(* CoDeSys 2.3.9.42 project: A100-60_CR0020_V050003.pro *)
(* Libraries: ifm_CR0020\ifm_CR0020_V050003.lib 15.12.08 18:14:24, Util.lib 6.11.07 15:39:24, standard.lib 4.10.05 11:14:46, ifm_J1939\ifm_CAN1_EXT_V050008.lib 12.9.08 16:16:28, ifm_J1939\ifm_J1939_1_V050008.lib 5.2.08 18:55:26, ifm_J1939\ifm_J1939_2_V050008.lib 5.2.08 18:56:24 *)

(* PLC configuration (modules and I/O channels)
Inputs Port0 [Eingangsport0] node 0, in %IB0 out %QB0
  I00 AT %IX0.0 [BoolChannelIn] Connector 1, Pin 08, (see Configuration Byte I00_MODE)
  I01 AT %IX0.1 [BoolChannelIn] Connector 1, Pin 27, (see Configuration Byte I01_MODE)
  I02 AT %IX0.2 [BoolChannelIn] Connector 1, Pin 09, (see Configuration Byte I02_MODE)
  I03 AT %IX0.3 [BoolChannelIn] Connector 1, Pin 28, (see Configuration Byte I03_MODE)
  I04 AT %IX0.4 [BoolChannelIn] Connector 1, Pin 10, (see Configuration Byte I04_MODE)
  I05 AT %IX0.5 [BoolChannelIn] Connector 1, Pin 29, (see Configuration Byte I05_MODE)
  I06 AT %IX0.6 [BoolChannelIn] Connector 1, Pin 11, (see Configuration Byte I06_MODE)
  I07 AT %IX0.7 [BoolChannelIn] Connector 1, Pin 30, (see Configuration Byte I07_MODE)
Inputs Port1 [Eingangsport1] node 0, in %IB1 out %QB0
  I10 AT %IX0.8 [BoolChannelIn] Connector 1, Pin 44, (see Configuration Byte I10_MODE)
  I11 AT %IX0.9 [BoolChannelIn] Connector 1, Pin 45, (see Configuration Byte I11_MODE)
  I12 AT %IX0.10 [BoolChannelIn] Connector 1, Pin 46, (see Configuration Byte I12_MODE)
  I13 AT %IX0.11 [BoolChannelIn] Connector 1, Pin 47, (see Configuration Byte I13_MODE)
  I14 AT %IX0.12 [BoolChannelIn] Connector 1, Pin 20, (see Configuration Byte I14_MODE)
  I15 AT %IX0.13 [BoolChannelIn] Connector 1, Pin 02, (see Configuration Byte I15_MODE)
  I16 AT %IX0.14 [BoolChannelIn] Connector 1, Pin 21, (see Configuration Byte I16_MODE)
  I17 AT %IX0.15 [BoolChannelIn] Connector 1, Pin 38, (see Configuration Byte I17_MODE)
Inputs Port2 [Eingangsport2] node 0, in %IB2 out %QB0
  I20 AT %IX1.0 [BoolChannelIn] Connector 1, Pin 36, (see Configuration Byte I20_MODE)
  I21 AT %IX1.1 [BoolChannelIn] Connector 1, Pin 54, (see Configuration Byte I21_MODE)
  I22 AT %IX1.2 [BoolChannelIn] Connector 1, Pin 17, (see Configuration Byte I22_MODE)
  I23 AT %IX1.3 [BoolChannelIn] Connector 1, Pin 53, (see Configuration Byte I23_MODE)
  I24 AT %IX1.4 [BoolChannelIn] Connector 1, Pin 19, (see Configuration Byte I24_MODE)
  I25 AT %IX1.5 [BoolChannelIn] Connector 1, Pin 55, (see Configuration Byte I25_MODE)
  I26 AT %IX1.6 [BoolChannelIn] Connector 1, Pin 18, (see Configuration Byte I26_MODE)
  I27 AT %IX1.7 [BoolChannelIn] Connector 1, Pin 37, (see Configuration Byte I27_MODE)
Inputs Port3 [Eingangsport3] node 0, in %IB3 out %QB0
  I30 AT %IX1.8 [BoolChannelIn] Connector 1, Pin 39, (see Configuration Byte I30_MODE)
  I31 AT %IX1.9 [BoolChannelIn] Connector 1, Pin 03, (see Configuration Byte I31_MODE)
  I32 AT %IX1.10 [BoolChannelIn] Connector 1, Pin 40, (see Configuration Byte I32_MODE)
  I33 AT %IX1.11 [BoolChannelIn] Connector 1, Pin 22, (see Configuration Byte I33_MODE)
  I34 AT %IX1.12 [BoolChannelIn] Connector 1, Pin 41, (see Configuration Byte I34_MODE)
  I35 AT %IX1.13 [BoolChannelIn] Connector 1, Pin 42, (see Configuration Byte I35_MODE)
  I36 AT %IX1.14 [BoolChannelIn] Connector 1, Pin 43, (see Configuration Byte I36_MODE)
  I37 AT %IX1.15 [BoolChannelIn] Connector 1, Pin 04, (see Configuration Byte I37_MODE)
Inputs Port4 [Eingangsport4] node 0, in %IB4 out %QB0
  I40 AT %IX2.0 [BoolChannelIn] Connector 1, Pin 48, (see Configuration Byte I40_MODE)
  I41 AT %IX2.1 [BoolChannelIn] Connector 1, Pin 49, (see Configuration Byte I41_MODE)
  I42 AT %IX2.2 [BoolChannelIn] Connector 1, Pin 31, (see Configuration Byte I42_MODE)
  I43 AT %IX2.3 [BoolChannelIn] Connector 1, Pin 50, (see Configuration Byte I43_MODE)
  I44 AT %IX2.4 [BoolChannelIn] Connector 1, Pin 51, (see Configuration Byte I44_MODE)
  I45 AT %IX2.5 [BoolChannelIn] Connector 1, Pin 52, (see Configuration Byte I45_MODE)
  I46 AT %IX2.6 [BoolChannelIn] Connector 1, Pin 16, (see Configuration Byte I46_MODE)
  I47 AT %IX2.7 [BoolChannelIn] Connector 1, Pin 35, (see Configuration Byte I47_MODE)
ANALOG0 AT %IW3 [WordChannelIn] Connector 1, Pin 08, ANALOG CHANNEL 0
ANALOG1 AT %IW4 [WordChannelIn] Connector 1, Pin 27, ANALOG CHANNEL 1
ANALOG2 AT %IW5 [WordChannelIn] Connector 1, Pin 09, ANALOG CHANNEL 2
ANALOG3 AT %IW6 [WordChannelIn] Connector 1, Pin 28, ANALOG CHANNEL 3
ANALOG4 AT %IW7 [WordChannelIn] Connector 1, Pin 10, ANALOG CHANNEL 4
ANALOG5 AT %IW8 [WordChannelIn] Connector 1, Pin 29, ANALOG CHANNEL 5
ANALOG6 AT %IW9 [WordChannelIn] Connector 1, Pin 11, ANALOG CHANNEL 6
ANALOG7 AT %IW10 [WordChannelIn] Connector 1, Pin 30, ANALOG CHANNEL 7
Inputs Miscellaneous [Eingaenge] node 0, in %IB22 out %QB0
  SUPPLY_VOLTAGE AT %IW11 [WordChannelIn] SUPPLY VOLTAGE
  CLAMP_15 AT %IX12.0 [WordChannelIn] CLAMP 15
Outputs Port1 [Ausgangsport1] node 0, in %IB64 out %QB0
  Q10 AT %QX0.0 [BoolChannelOut] Connector 1, Pin 44, (see Configuration Byte Q10_MODE)
  Q11 AT %QX0.1 [BoolChannelOut] Connector 1, Pin 45, (see Configuration Byte Q11_MODE)
  Q12 AT %QX0.2 [BoolChannelOut] Connector 1, Pin 46, (see Configuration Byte Q12_MODE)
  Q13 AT %QX0.3 [BoolChannelOut] Connector 1, Pin 47, (see Configuration Byte Q13_MODE)
Outputs Port2 [Ausgangsport2] node 0, in %IB64 out %QB0
  Q20 AT %QX0.4 [BoolChannelOut] Connector 1, Pin 36, (see Configuration Byte Q20_MODE)
  Q21 AT %QX0.5 [BoolChannelOut] Connector 1, Pin 54, (see Configuration Byte Q21_MODE)
  Q22 AT %QX0.6 [BoolChannelOut] Connector 1, Pin 17, (see Configuration Byte Q22_MODE)
  Q23 AT %QX0.7 [BoolChannelOut] Connector 1, Pin 53, (see Configuration Byte Q23_MODE)
Outputs Port3 [Ausgangsport3] node 0, in %IB64 out %QB1
  Q30 AT %QX0.8 [BoolChannelOut] Connector 1, Pin 39, (see Configuration Byte Q30_MODE)
  Q31 AT %QX0.9 [BoolChannelOut] Connector 1, Pin 03, (see Configuration Byte Q31_MODE)
  Q32 AT %QX0.10 [BoolChannelOut] Connector 1, Pin 40, (see Configuration Byte Q32_MODE)
  Q33 AT %QX0.11 [BoolChannelOut] Connector 1, Pin 22, (see Configuration Byte Q33_MODE)
  Q34 AT %QX0.12 [BoolChannelOut] Connector 1, Pin 41, (see Configuration Byte Q34_MODE)
  Q35 AT %QX0.13 [BoolChannelOut] Connector 1, Pin 42, (see Configuration Byte Q35_MODE)
  Q36 AT %QX0.14 [BoolChannelOut] Connector 1, Pin 43, (see Configuration Byte Q36_MODE)
  Q37 AT %QX0.15 [BoolChannelOut] Connector 1, Pin 04, (see Configuration Byte Q37_MODE)
Outputs Port4 [Ausgangsport4] node 0, in %IB64 out %QB2
  Q40 AT %QX1.0 [BoolChannelOut] Connector 1, Pin 48, (see Configuration Byte Q40_MODE)
  Q41 AT %QX1.1 [BoolChannelOut] Connector 1, Pin 49, (see Configuration Byte Q41_MODE)
  Q42 AT %QX1.2 [BoolChannelOut] Connector 1, Pin 31, (see Configuration Byte Q42_MODE)
  Q43 AT %QX1.3 [BoolChannelOut] Connector 1, Pin 50, (see Configuration Byte Q43_MODE)
  Q44 AT %QX1.4 [BoolChannelOut] Connector 1, Pin 51, (see Configuration Byte Q44_MODE)
  Q45 AT %QX1.5 [BoolChannelOut] Connector 1, Pin 52, (see Configuration Byte Q45_MODE)
  Q46 AT %QX1.6 [BoolChannelOut] Connector 1, Pin 16, (see Configuration Byte Q46_MODE)
  Q47 AT %QX1.7 [BoolChannelOut] Connector 1, Pin 35, (see Configuration Byte Q47_MODE)
Input Modes Port0 [EingangsModi0] node 0, in %IB64 out %QB8
  I00_MODE AT %QB8 [ByteChannelOut] Configuration Byte for Input Pin 08, Connector 1
  I01_MODE AT %QB9 [ByteChannelOut] Configuration Byte for Input Pin 27, Connector 1
  I02_MODE AT %QB10 [ByteChannelOut] Configuration Byte for Input Pin 09, Connector 1
  I03_MODE AT %QB11 [ByteChannelOut] Configuration Byte for Input Pin 28, Connector 1
  I04_MODE AT %QB12 [ByteChannelOut] Configuration Byte for Input Pin 10, Connector 1
  I05_MODE AT %QB13 [ByteChannelOut] Configuration Byte for Input Pin 29, Connector 1
  I06_MODE AT %QB14 [ByteChannelOut] Configuration Byte for Input Pin 11, Connector 1
  I07_MODE AT %QB15 [ByteChannelOut] Configuration Byte for Input Pin 30, Connector 1
Input Modes Port1 [EingangsModi1] node 0, in %IB64 out %QB16
  I14_MODE AT %QB16 [ByteChannelOut] Configuration Byte for Input Pin 20, Connector 1
  I15_MODE AT %QB17 [ByteChannelOut] Configuration Byte for Input Pin 02, Connector 1
  I16_MODE AT %QB18 [ByteChannelOut] Configuration Byte for Input Pin 21, Connector 1
  I17_MODE AT %QB19 [ByteChannelOut] Configuration Byte for Input Pin 38, Connector 1
Input Modes Port2 [EingangsModi2] node 0, in %IB64 out %QB20
  I24_MODE AT %QB20 [ByteChannelOut] Configuration Byte for Input Pin 19, Connector 1
  I25_MODE AT %QB21 [ByteChannelOut] Configuration Byte for Input Pin 55, Connector 1
  I26_MODE AT %QB22 [ByteChannelOut] Configuration Byte for Input Pin 18, Connector 1
  I27_MODE AT %QB23 [ByteChannelOut] Configuration Byte for Input Pin 37, Connector 1
Input Modes Port3 [EingangsModi3] node 0, in %IB64 out %QB24
  I30_MODE AT %QB24 [ByteChannelOut] Configuration Byte for Input Pin 39, Connector 1
  I31_MODE AT %QB25 [ByteChannelOut] Configuration Byte for Input Pin 03, Connector 1
  I32_MODE AT %QB26 [ByteChannelOut] Configuration Byte for Input Pin 40, Connector 1
  I33_MODE AT %QB27 [ByteChannelOut] Configuration Byte for Input Pin 22, Connector 1
  I34_MODE AT %QB28 [ByteChannelOut] Configuration Byte for Input Pin 41, Connector 1
  I35_MODE AT %QB29 [ByteChannelOut] Configuration Byte for Input Pin 42, Connector 1
  I36_MODE AT %QB30 [ByteChannelOut] Configuration Byte for Input Pin 43, Connector 1
  I37_MODE AT %QB31 [ByteChannelOut] Configuration Byte for Input Pin 04, Connector 1
Input Modes Port4 [EingangsModi4] node 0, in %IB64 out %QB32
  I40_MODE AT %QB32 [ByteChannelOut] Configuration Byte for Input Pin 48, Connector 1
  I41_MODE AT %QB33 [ByteChannelOut] Configuration Byte for Input Pin 49, Connector 1
  I42_MODE AT %QB34 [ByteChannelOut] Configuration Byte for Input Pin 31, Connector 1
  I43_MODE AT %QB35 [ByteChannelOut] Configuration Byte for Input Pin 50, Connector 1
  I44_MODE AT %QB36 [ByteChannelOut] Configuration Byte for Input Pin 51, Connector 1
  I45_MODE AT %QB37 [ByteChannelOut] Configuration Byte for Input Pin 52, Connector 1
  I46_MODE AT %QB38 [ByteChannelOut] Configuration Byte for Input Pin 16, Connector 1
  I47_MODE AT %QB39 [ByteChannelOut] Configuration Byte for Input Pin 35, Connector 1
Output Modes Port1 [AusgangsModi1] node 0, in %IB64 out %QB40
  Q10_MODE AT %QB40 [ByteChannelOut] Configuration Byte for Output Pin 44, Connector 1
  Q11_MODE AT %QB41 [ByteChannelOut] Configuration Byte for Output Pin 45, Connector 1
  Q12_MODE AT %QB42 [ByteChannelOut] Configuration Byte for Output Pin 46, Connector 1
  Q13_MODE AT %QB43 [ByteChannelOut] Configuration Byte for Output Pin 47, Connector 1
Output Modes Port2 [AusgangsModi2] node 0, in %IB64 out %QB44
  Q20_MODE AT %QB44 [ByteChannelOut] Configuration Byte for Output Pin 36, Connector 1
  Q21_MODE AT %QB45 [ByteChannelOut] Configuration Byte for Output Pin 54, Connector 1
  Q22_MODE AT %QB46 [ByteChannelOut] Configuration Byte for Output Pin 17, Connector 1
  Q23_MODE AT %QB47 [ByteChannelOut] Configuration Byte for Output Pin 53, Connector 1
Output Modes Port3 [AusgangsModi3] node 0, in %IB64 out %QB48
  Q30_MODE AT %QB48 [ByteChannelOut] Configuration Byte for Output Pin 39, Connector 1
  Q31_MODE AT %QB49 [ByteChannelOut] Configuration Byte for Output Pin 03, Connector 1
  Q32_MODE AT %QB50 [ByteChannelOut] Configuration Byte for Output Pin 40, Connector 1
  Q33_MODE AT %QB51 [ByteChannelOut] Configuration Byte for Output Pin 22, Connector 1
  Q34_MODE AT %QB52 [ByteChannelOut] Configuration Byte for Output Pin 41, Connector 1
  Q35_MODE AT %QB53 [ByteChannelOut] Configuration Byte for Output Pin 42, Connector 1
  Q36_MODE AT %QB54 [ByteChannelOut] Configuration Byte for Output Pin 43, Connector 1
  Q37_MODE AT %QB55 [ByteChannelOut] Configuration Byte for Output Pin 04, Connector 1
Output Modes Port4 [AusgangsModi4] node 0, in %IB64 out %QB56
  Q40_MODE AT %QB56 [ByteChannelOut] Configuration Byte for Output Pin 48, Connector 1
  Q41_MODE AT %QB57 [ByteChannelOut] Configuration Byte for Output Pin 49, Connector 1
  Q42_MODE AT %QB58 [ByteChannelOut] Configuration Byte for Output Pin 31, Connector 1
  Q43_MODE AT %QB59 [ByteChannelOut] Configuration Byte for Output Pin 50, Connector 1
  Q44_MODE AT %QB60 [ByteChannelOut] Configuration Byte for Output Pin 51, Connector 1
  Q45_MODE AT %QB61 [ByteChannelOut] Configuration Byte for Output Pin 52, Connector 1
  Q46_MODE AT %QB62 [ByteChannelOut] Configuration Byte for Output Pin 16, Connector 1
  Q47_MODE AT %QB63 [ByteChannelOut] Configuration Byte for Output Pin 35, Connector 1
*)

(* Global variable list: GV_CAL *)
VAR_GLOBAL
(*
	Аналоговый - aChannel_ADC - adc := 0 - 16
	Частотный  - aChannel_PIN - pin := 1 - 8
	ШИМ        - aChannel_PWM - pwm := 2 - 8
	ПИД        - aChannel_PID - pid := 3 - 8
	Энкодер    - aChannel_ENC - enc := 4 - 8
	Расчет     - aChannel_FRM - frm := 5 - 8
	Расход                          := 6 - 8
*)

(*Максимальный размер массива параметров каналов*)
	iSizeArrayParamMax : INT := 64;

(**)
	aPage_Channel      : ARRAY [0..63] OF Page_Channel;(**)

(*Переменные выбора текущего режима работы*)
	dwCurrMode         : DWORD := 1;(*Текущий режим работы установки*)
	bCurrModeChange    : BOOL  := 0;(*Флаг смены текущего режима работы установки*)

(*Переменные каналов ШИМ*)
	rArrayDataPWM_XH      : ARRAY [1..8] OF REAL;(**)
	rArrayDataPWM_XL      : ARRAY [1..8] OF REAL;(**)
	rArrayDataPWM_YH      : ARRAY [1..8] OF REAL;(**)
	rArrayDataPWM_YL      : ARRAY [1..8] OF REAL;(**)
	dwArrayAverTimePWM    : ARRAY [1..8] OF DWORD;(*Времена усреднения каналов*)
	rArrayDataPWM_DZ_MAX  : ARRAY [1..8] OF REAL;(*Коэффициенты, учитывающие особенности механики*)
	dwArrayDataPWM_DZ_MIN : ARRAY [1..8] OF DWORD;(**)

	dwArrayNumberPWM      : ARRAY [1..8] OF DWORD;(**)
	rArrayParam10PWM      : ARRAY [1..8] OF REAL;(**)

(*Переменные каналов ПИД*)
	rArrayDataPID_P_Coef  : ARRAY [1..8] OF REAL;(**)
	rArrayDataPID_I_Coef  : ARRAY [1..8] OF REAL;(**)
	rArrayDataPID_D_Coef  : ARRAY [1..8] OF REAL;(**)
	rArrayDataPID_Shift   : ARRAY [1..8] OF REAL;(**)
	dwArrayAverTimePID    : ARRAY [1..8] OF DWORD;(*Времена усреднения каналов*)
	rArrayCoeffPID        : ARRAY [1..8] OF REAL;(*Коэффициенты, учитывающие особенности механики*)
	dwArrayDescriptPID    : ARRAY [1..8] OF DWORD;(**)

	dwArrayNumberPID      : ARRAY [1..8] OF DWORD;(**)
	rArrayParam10PID      : ARRAY [1..8] OF REAL;(**)
END_VAR

(* Global variable list: GV_CAN1_J1939 *)
VAR_GLOBAL
(*Переменные параметров CAN шины*)
	byCAN1_PCUnitID            : BYTE := 16#01;(*ID компьютерной панели, подключенной на CAN1*)

	byCAN1_DownloadID          : BYTE := 127;(*ID контроллера CAN1 (Download)*)
	byCAN1_PreferAddr          : BYTE := 16#40;(**)             byCurrCAN1Addr   : BYTE;(*Текущий адрес на шине CAN PC*)
	byCAN1_Channel             : BYTE := 1;
	byCAN1_DataLength          : BYTE := 8;(*Количество байт в пакете CAN1*)
	wCAN1_BaudRate             : WORD := 250;(*Скорость передачи данных 250 кбит/сек*)
	bCAN1_TransmitEnable       : BOOL := 1;(*Разрешение работы CAN1 на передачу*)

	bCAN1_J1939NotActive       : BOOL := 0;(*CAN J1939 Not active*)
	bCAN1_J1939Errors          : BOOL := 0;(*CAN J1939 Signalling of errors*)

(*Переменные приема в CAN J1939*)
	CAN1RX_UNIT_ADDR           : J1939_1_RECEIVE;  abyCAN1RX_UNIT_ADDR           : ARRAY [0..7] OF BYTE;

	CAN1RX_CHANNEL_INDEX       : J1939_1_RECEIVE;  abyCAN1RX_CHANNEL_INDEX       : ARRAY [0..7] OF BYTE;
	CAN1RX_PARAM00             : J1939_1_RECEIVE;  abyCAN1RX_PARAM00             : ARRAY [0..7] OF BYTE;
	CAN1RX_PARAM01             : J1939_1_RECEIVE;  abyCAN1RX_PARAM01             : ARRAY [0..7] OF BYTE;
	CAN1RX_PARAM02             : J1939_1_RECEIVE;  abyCAN1RX_PARAM02             : ARRAY [0..7] OF BYTE;
	CAN1RX_PARAM03             : J1939_1_RECEIVE;  abyCAN1RX_PARAM03             : ARRAY [0..7] OF BYTE;
	CAN1RX_PARAM04             : J1939_1_RECEIVE;  abyCAN1RX_PARAM04             : ARRAY [0..7] OF BYTE;
	CAN1RX_PARAM05             : J1939_1_RECEIVE;  abyCAN1RX_PARAM05             : ARRAY [0..7] OF BYTE;
	CAN1RX_PARAM06             : J1939_1_RECEIVE;  abyCAN1RX_PARAM06             : ARRAY [0..7] OF BYTE;
	CAN1RX_PARAM07             : J1939_1_RECEIVE;  abyCAN1RX_PARAM07             : ARRAY [0..7] OF BYTE;
	CAN1RX_PARAM08             : J1939_1_RECEIVE;  abyCAN1RX_PARAM08             : ARRAY [0..7] OF BYTE;
	CAN1RX_PARAM09             : J1939_1_RECEIVE;  abyCAN1RX_PARAM09             : ARRAY [0..7] OF BYTE;
	CAN1RX_PARAM10             : J1939_1_RECEIVE;  abyCAN1RX_PARAM10             : ARRAY [0..7] OF BYTE;

	CAN1RX_CURR_MODE           : J1939_1_RECEIVE;  abyCAN1RX_CURR_MODE           : ARRAY [0..7] OF BYTE;
	CAN1RX_COMMAND             : J1939_1_RECEIVE;  abyCAN1RX_COMMAND             : ARRAY [0..7] OF BYTE;

	CAN1RX_Set_GN2TempManual   : J1939_1_RECEIVE;  abyCAN1RX_Set_GN2TempManual   : ARRAY [0..7] OF BYTE;
	CAN1RX_Set_GN2OverPres     : J1939_1_RECEIVE;  abyCAN1RX_Set_GN2OverPres     : ARRAY [0..7] OF BYTE;
	CAN1RX_Set_BoostPresManual : J1939_1_RECEIVE;  abyCAN1RX_Set_BoostPresManual : ARRAY [0..7] OF BYTE;
	CAN1RX_Set_GN2Rate         : J1939_1_RECEIVE;  abyCAN1RX_Set_GN2Rate         : ARRAY [0..7] OF BYTE;
	CAN1RX_Set_LN2SaturTemp    : J1939_1_RECEIVE;  abyCAN1RX_Set_LN2SaturTemp    : ARRAY [0..7] OF BYTE;

(*Переменные отправки в CAN J1939. Используемые PGN*)
	CAN1TX_UNIT_ADDR           : J1939_1_TRANSMIT; abyCAN1TX_UNIT_ADDR           : ARRAY [0..7] OF BYTE; dwPGN1_UNIT_ADDR           : DWORD := 16#F000;

	CAN1TX_CHANNEL_INDEX       : J1939_1_TRANSMIT; abyCAN1TX_CHANNEL_INDEX       : ARRAY [0..7] OF BYTE; dwPGN1_CHANNEL_INDEX       : DWORD := 16#F001;
	CAN1TX_PARAM00             : J1939_1_TRANSMIT; abyCAN1TX_PARAM00             : ARRAY [0..7] OF BYTE; dwPGN1_PARAM00             : DWORD := 16#F002;
	CAN1TX_PARAM01             : J1939_1_TRANSMIT; abyCAN1TX_PARAM01             : ARRAY [0..7] OF BYTE; dwPGN1_PARAM01             : DWORD := 16#F003;
	CAN1TX_PARAM02             : J1939_1_TRANSMIT; abyCAN1TX_PARAM02             : ARRAY [0..7] OF BYTE; dwPGN1_PARAM02             : DWORD := 16#F004;
	CAN1TX_PARAM03             : J1939_1_TRANSMIT; abyCAN1TX_PARAM03             : ARRAY [0..7] OF BYTE; dwPGN1_PARAM03             : DWORD := 16#F005;
	CAN1TX_PARAM04             : J1939_1_TRANSMIT; abyCAN1TX_PARAM04             : ARRAY [0..7] OF BYTE; dwPGN1_PARAM04             : DWORD := 16#F006;
	CAN1TX_PARAM05             : J1939_1_TRANSMIT; abyCAN1TX_PARAM05             : ARRAY [0..7] OF BYTE; dwPGN1_PARAM05             : DWORD := 16#F007;
	CAN1TX_PARAM06             : J1939_1_TRANSMIT; abyCAN1TX_PARAM06             : ARRAY [0..7] OF BYTE; dwPGN1_PARAM06             : DWORD := 16#F008;
	CAN1TX_PARAM07             : J1939_1_TRANSMIT; abyCAN1TX_PARAM07             : ARRAY [0..7] OF BYTE; dwPGN1_PARAM07             : DWORD := 16#F009;
	CAN1TX_PARAM08             : J1939_1_TRANSMIT; abyCAN1TX_PARAM08             : ARRAY [0..7] OF BYTE; dwPGN1_PARAM08             : DWORD := 16#F00A;
	CAN1TX_PARAM09             : J1939_1_TRANSMIT; abyCAN1TX_PARAM09             : ARRAY [0..7] OF BYTE; dwPGN1_PARAM09             : DWORD := 16#F00B;
	CAN1TX_PARAM10             : J1939_1_TRANSMIT; abyCAN1TX_PARAM10             : ARRAY [0..7] OF BYTE; dwPGN1_PARAM10             : DWORD := 16#F00C;

	CAN1TX_CURR_MODE           : J1939_1_TRANSMIT; abyCAN1TX_CURR_MODE           : ARRAY [0..7] OF BYTE; dwPGN1_CURR_MODE           : DWORD := 16#F00D;

	CAN1TX_TOTAL_TIME          : J1939_1_TRANSMIT; abyCAN1TX_TOTAL_TIME          : ARRAY [0..7] OF BYTE; dwPGN1_TOTAL_TIME          : DWORD := 16#F00E;
	CAN1TX_LAST_TIME           : J1939_1_TRANSMIT; abyCAN1TX_LAST_TIME           : ARRAY [0..7] OF BYTE; dwPGN1_LAST_TIME           : DWORD := 16#F00F;

	CAN1TX_COMMAND             : J1939_1_TRANSMIT; abyCAN1TX_COMMAND             : ARRAY [0..7] OF BYTE; dwPGN1_COMMAND             : DWORD := 16#F010;

	CAN1TX_STATE_ADC_MS        : J1939_1_TRANSMIT; abyCAN1TX_STATE_ADC_MS        : ARRAY [0..7] OF BYTE; dwPGN1_STATE_ADC_MS        : DWORD := 16#F011;
	CAN1TX_STATE_ADC_SL1       : J1939_1_TRANSMIT; abyCAN1TX_STATE_ADC_SL1       : ARRAY [0..7] OF BYTE; dwPGN1_STATE_ADC_SL1       : DWORD := 16#F012;
	CAN1TX_STATE_ADC_SL2       : J1939_1_TRANSMIT; abyCAN1TX_STATE_ADC_SL2       : ARRAY [0..7] OF BYTE; dwPGN1_STATE_ADC_SL2       : DWORD := 16#F013;
	CAN1TX_STATE_ADC_SL3       : J1939_1_TRANSMIT; abyCAN1TX_STATE_ADC_SL3       : ARRAY [0..7] OF BYTE; dwPGN1_STATE_ADC_SL3       : DWORD := 16#F014;

	CAN1TX_MS_SV               : J1939_1_TRANSMIT; abyCAN1TX_MS_SV               : ARRAY [0..7] OF BYTE; dwPGN1_MS_SV               : DWORD := 16#F015;
	CAN1TX_MS_T                : J1939_1_TRANSMIT; abyCAN1TX_MS_T                : ARRAY [0..7] OF BYTE; dwPGN1_MS_T                : DWORD := 16#F016;
	CAN1TX_PROG_CRC_MS         : J1939_1_TRANSMIT; abyCAN1TX_PROG_CRC_MS         : ARRAY [0..7] OF BYTE; dwPGN1_PROG_CRC_MS         : DWORD := 16#F017;
	CAN1TX_PROG_ID_MS          : J1939_1_TRANSMIT; abyCAN1TX_PROG_ID_MS          : ARRAY [0..7] OF BYTE; dwPGN1_PROG_ID_MS          : DWORD := 16#F018;

	CAN1TX_STATE_MS            : J1939_1_TRANSMIT; abyCAN1TX_STATE_MS            : ARRAY [0..7] OF BYTE; dwPGN1_STATE_MS            : DWORD := 16#F019;
	CAN1TX_STATE_SL1           : J1939_1_TRANSMIT; abyCAN1TX_STATE_SL1           : ARRAY [0..7] OF BYTE; dwPGN1_STATE_SL1           : DWORD := 16#F01A;
	CAN1TX_STATE_SL2           : J1939_1_TRANSMIT; abyCAN1TX_STATE_SL2           : ARRAY [0..7] OF BYTE; dwPGN1_STATE_SL2           : DWORD := 16#F01B;
	CAN1TX_STATE_SL3           : J1939_1_TRANSMIT; abyCAN1TX_STATE_SL3           : ARRAY [0..7] OF BYTE; dwPGN1_STATE_SL3           : DWORD := 16#F01C;

	CAN1TX_DM1                 : J1939_1_TRANSMIT; abyCAN1TX_DM1                 : ARRAY [0..7] OF BYTE; dwPGN1_DM1                 : DWORD := 16#F01D;
	CAN1TX_DM2                 : J1939_1_TRANSMIT; abyCAN1TX_DM2                 : ARRAY [0..7] OF BYTE; dwPGN1_DM2                 : DWORD := 16#F01E;
	CAN1TX_DM1_DESCR           : J1939_1_TRANSMIT; abyCAN1TX_DM1_DESCR           : ARRAY [0..7] OF BYTE; dwPGN1_DM1_DESCR           : DWORD := 16#F01F;
	CAN1TX_DM2_DESCR           : J1939_1_TRANSMIT; abyCAN1TX_DM2_DESCR           : ARRAY [0..7] OF BYTE; dwPGN1_DM2_DESCR           : DWORD := 16#F020;

	CAN1TX_GN2_Temp            : J1939_1_TRANSMIT; abyCAN1TX_GN2_Temp            : ARRAY [0..7] OF BYTE; dwPGN1_GN2_Temp            : DWORD := 16#F03F;
	CAN1TX_WF_PresOut          : J1939_1_TRANSMIT; abyCAN1TX_WF_PresOut          : ARRAY [0..7] OF BYTE; dwPGN1_WF_PresOut          : DWORD := 16#F040;
	CAN1TX_LN2_Temp            : J1939_1_TRANSMIT; abyCAN1TX_LN2_Temp            : ARRAY [0..7] OF BYTE; dwPGN1_LN2_Temp            : DWORD := 16#F03D;
	CAN1TX_BoostPres           : J1939_1_TRANSMIT; abyCAN1TX_BoostPres           : ARRAY [0..7] OF BYTE; dwPGN1_BoostPres           : DWORD := 16#F03C;
	CAN1TX_HydHeatPres         : J1939_1_TRANSMIT; abyCAN1TX_HydHeatPres         : ARRAY [0..7] OF BYTE; dwPGN1_HydHeatPres         : DWORD := 16#F041;
	CAN1TX_CoolTempIn          : J1939_1_TRANSMIT; abyCAN1TX_CoolTempIn          : ARRAY [0..7] OF BYTE; dwPGN1_CoolTempIn          : DWORD := 16#F042;

	CAN1TX_TriplexRPM          : J1939_1_TRANSMIT; abyCAN1TX_TriplexRPM          : ARRAY [0..7] OF BYTE; dwPGN1_TriplexRPM          : DWORD := 16#F046;

	CAN1TX_InputState          : J1939_1_TRANSMIT; abyCAN1TX_InputState          : ARRAY [0..7] OF BYTE; dwPGN1_InputState          : DWORD := 16#F047;
	CAN1TX_OutputState         : J1939_1_TRANSMIT; abyCAN1TX_OutputState         : ARRAY [0..7] OF BYTE; dwPGN1_OutputState         : DWORD := 16#F048;

	CAN1TX_Current_GN2Rate     : J1939_1_TRANSMIT; abyCAN1TX_Current_GN2Rate     : ARRAY [0..7] OF BYTE; dwPGN1_Current_GN2Rate     : DWORD := 16#F049;
	CAN1TX_TotalAmountGN2      : J1939_1_TRANSMIT; abyCAN1TX_TotalAmountGN2      : ARRAY [0..7] OF BYTE; dwPGN1_TotalAmountGN2      : DWORD := 16#F04A;
	CAN1TX_CurrEngineRPM       : J1939_1_TRANSMIT; abyCAN1TX_CurrEngineRPM       : ARRAY [0..7] OF BYTE; dwPGN1_CurrEngineRPM       : DWORD := 16#F04B;
	CAN1TX_CurrNumberGear      : J1939_1_TRANSMIT; abyCAN1TX_CurrNumberGear      : ARRAY [0..7] OF BYTE; dwPGN1_CurrNumberGear      : DWORD := 16#F04C;
	CAN1TX_Set_GN2TempManual   : J1939_1_TRANSMIT; abyCAN1TX_Set_GN2TempManual   : ARRAY [0..7] OF BYTE; dwPGN1_Set_GN2TempManual   : DWORD := 16#F04D;
	CAN1TX_Set_GN2OverPres     : J1939_1_TRANSMIT; abyCAN1TX_Set_GN2OverPres     : ARRAY [0..7] OF BYTE; dwPGN1_Set_GN2OverPres     : DWORD := 16#F04E;
	CAN1TX_Set_BoostPresManual : J1939_1_TRANSMIT; abyCAN1TX_Set_BoostPresManual : ARRAY [0..7] OF BYTE; dwPGN1_Set_BoostPresManual : DWORD := 16#F04F;
	CAN1TX_Set_GN2Rate         : J1939_1_TRANSMIT; abyCAN1TX_Set_GN2Rate         : ARRAY [0..7] OF BYTE; dwPGN1_Set_GN2Rate         : DWORD := 16#F050;
	CAN1TX_Set_LN2SaturTemp    : J1939_1_TRANSMIT; abyCAN1TX_Set_LN2SaturTemp    : ARRAY [0..7] OF BYTE; dwPGN1_Set_LN2SaturTemp    : DWORD := 16#F051;
	CAN1TX_ReqStageOper        : J1939_1_TRANSMIT; abyCAN1TX_ReqStageOper        : ARRAY [0..7] OF BYTE; dwPGN1_ReqStageOper        : DWORD := 16#F052;
	CAN1TX_CurStageOper        : J1939_1_TRANSMIT; abyCAN1TX_CurStageOper        : ARRAY [0..7] OF BYTE; dwPGN1_CurStageOper        : DWORD := 16#F053;

	CAN1TX_ErrorState          : J1939_1_TRANSMIT; abyCAN1TX_ErrorState          : ARRAY [0..7] OF BYTE; dwPGN1_ErrorState          : DWORD := 16#F054;
	CAN1TX_ProcessState        : J1939_1_TRANSMIT; abyCAN1TX_ProcessState        : ARRAY [0..7] OF BYTE; dwPGN1_ProcessState        : DWORD := 16#F055;
	CAN1TX_GN2_Pres            : J1939_1_TRANSMIT; abyCAN1TX_GN2_Pres            : ARRAY [0..7] OF BYTE; dwPGN1_GN2_Pres            : DWORD := 16#F056;
	CAN1TX_CoolTempInMin       : J1939_1_TRANSMIT; abyCAN1TX_CoolTempInMin       : ARRAY [0..7] OF BYTE; dwPGN1_CoolTempInMin       : DWORD := 16#F057;

	dwCHANNEL_INDEX            : DWORD := 16#FFFF;(*Индекс текущего канала*)

	bCommand                   : BOOL := 0;(*Флаг получения новой команды*)
	diCommand                  : DINT := 0;(*Номер команды*)
END_VAR

(* Global variable list: GV_CAN2_J1939 *)
VAR_GLOBAL
(*Переменные параметров CAN шины*)
	wECUEngineAddress     : WORD := 16#0;(*The Engine ECU always assumes the fixed source address 0x00*)
	wECUAddress           : WORD := 16#3;(*The Transmission ECU always assumes the fixed source address 0x03*)

	byCAN2_DownloadID     : BYTE := 127;(*ID контроллера CAN2 (Download)*)
	byCAN2_PreferAddr     : BYTE := 16#29;(**)
	byCAN2_Channel        : BYTE := 2;
	byCAN2_DataLength     : BYTE := 8;(*Количество байт в пакете CAN2*)
	wCAN2_BaudRate        : WORD := 250;(*Скорость передачи данных 250 кбит/сек*)
	bCAN2_TransmitEnable  : BOOL := 1;(*Разрешение работы CAN2 на передачу*)

	bCAN2_J1939NotActive  : BOOL := 0;(*CAN J1939 Not active*)
	bCAN2_J1939Errors     : BOOL := 0;(*CAN J1939 Signalling of errors*)

	bResetErrorsECU       : BOOL := 0;(**)
	bResetErrorsECU1      : BOOL := 0;(**)
	bResetErrorsECU2      : BOOL := 0;(**)
	bResetErrorsBuf       : BOOL := 0;(**)

(*Переменные приема в CAN J1939*)
	CAN2RX_EEC1           : J1939_2_RECEIVE; abyCAN2_Receive_EEC1 : ARRAY [1..8] OF BYTE;
	CAN2RX_ETC1           : J1939_2_RECEIVE; abyCAN2_Receive_ETC1 : ARRAY [1..8] OF BYTE;
	CAN2RX_ETC2           : J1939_2_RECEIVE; abyCAN2_Receive_ETC2 : ARRAY [1..8] OF BYTE;
	CAN2RX_TC1            : J1939_2_RECEIVE; abyCAN2_Receive_TC1  : ARRAY [1..8] OF BYTE;

	CAN2RX_DM1            : J1939_2_RECEIVE; abyCAN2_Receive_DM1  : ARRAY [1..130] OF BYTE;
	CAN2RX_DM2            : J1939_2_RECEIVE; abyCAN2_Receive_DM2  : ARRAY [1..130] OF BYTE;

(*Переменные отправки в CAN J1939*)
	CAN2TX_TSC1           : J1939_2_TRANSMIT;  abyCAN2TX_TSC1     : ARRAY [1..8] OF BYTE; dwPGN2_TSC1     : DWORD := 16#0000;
	CAN2TX_CCVS           : J1939_2_TRANSMIT;  abyCAN2TX_CCVS     : ARRAY [1..8] OF BYTE; dwPGN2_CCVS     : DWORD := 16#FEF1;

	CAN2TX_RQST_PGN       : J1939_2_TRANSMIT;  abyCAN2TX_RQST_PGN : ARRAY [1..3] OF BYTE; dwPGN2_RQST_PGN : DWORD := 16#EA00;
	CAN2TX_DM3            : J1939_2_TRANSMIT;  abyCAN2TX_DM3      : ARRAY [1..8] OF BYTE; dwPGN2_DM3      : DWORD := 16#FECC;
	CAN2TX_DM22           : J1939_2_TRANSMIT;  abyCAN2TX_DM22     : ARRAY [1..8] OF BYTE; dwPGN2_DM22     : DWORD := 16#C300;
	CAN2TX_AC             : J1939_2_TRANSMIT;  abyCAN2TX_AC       : ARRAY [1..8] OF BYTE; dwPGN2_AC       : DWORD := 16#EEFF;

	diRequiredSpeedSet    : DINT := 16#FFFF;
	wCruiseControlSet     : WORD := 16#FFFF;

	adwErrors_SPN_FMI_DM1 : ARRAY [1..32] OF DWORD;
	adwErrors_SPN_FMI_DM2 : ARRAY [1..32] OF DWORD;

	byErrorsQty_DM1       : BYTE := 0;
	byErrorsQty_DM2       : BYTE := 0;

	bEnableTransmit_DM1   : BOOL := 0;
	bEnableTransmit_DM2   : BOOL := 0;

	abyDataCurrentDM1     : ARRAY [1..8] OF BYTE;
	abyDataCurrentDM2     : ARRAY [1..8] OF BYTE;

	aCAN1ErrorDM1         : ARRAY [1..32] OF CAN1_ERROR_DM1;
	aCAN1ErrorDM2         : ARRAY [1..32] OF CAN1_ERROR_DM2;

	byLampStateDM1        : BYTE := 0;
	byLampStateDM2        : BYTE := 0;
END_VAR

VAR_GLOBAL CONSTANT
(*Electronic Engine Controller 1 - EEC1*)
	wPGN_EEC1                            : WORD := 61444;
	tRPT_EEC1                            : TIME := T#30ms;(*Transmission Repetition Rate*)     (*engine speed dependent*)
	byLEN_EEC1                           : BYTE := 8;(*Data Length (Number of bytes to be transmitted)*)
	byPG_EEC1                            : BYTE := 0;(*Data Page (Page address)*)
	byPDUFormat_EEC1                     : BYTE := 240;
	byPDUSpecific_EEC1                   : BYTE := 4;
	byPRIO_EEC1                          : BYTE := 3;(*Default Priority (Message priority)*)

	SPN_EngineSpeed                      : WORD := 190;(*Engine Speed*)

(*Electronic Transmission Controller 1 - ETC1*)
	wPGN_ETC1                            : WORD := 61442;
	tRPT_ETC1                            : TIME := T#0ms;(*Transmission Repetition Rate*)
	byLEN_ETC1                           : BYTE := 8;(*Data Length (Number of bytes to be transmitted)*)
	byPG_ETC1                            : BYTE := 0;(*Data Page (Page address)*)
	byPDUFormat_ETC1                     : BYTE := 240;
	byPDUSpecific_ETC1                   : BYTE := 2;
	byPRIO_ETC1                          : BYTE := 3;(*Default Priority (Message priority)*)

	SPN_TransmissionOutputShaftSpeed     : WORD := 191;(*Transmission Output Shaft Speed*)
	SPN_TransmissionInputShaftSpeed      : WORD := 161;(*Transmission Input Shaft Speed*)
	SPN_TransmissionTorqueConverterLockupClutchEngaged : WORD:=573;(*Transmission Torque Converter Lockup Clutch Engaged*)

(*Electronic Transmission Controller 2 - ETC2*)
	wPGN_ETC2                            : WORD := 61445;
	tRPT_ETC2                            : TIME := T#0ms;(*Transmission Repetition Rate*)
	byLEN_ETC2                           : BYTE := 8;(*Data Length (Number of bytes to be transmitted)*)
	byPG_ETC2                            : BYTE := 0;(*Data Page (Page address)*)
	byPDUFormat_ETC2                     : BYTE := 240;
	byPDUSpecific_ETC2                   : BYTE := 5;
	byPRIO_ETC2                          : BYTE := 6;(*Default Priority (Message priority)*)

	SPN_TransmissionSelectedGear         : WORD := 524;(*Transmission Selected Gear*)
	SPN_TransmissionCurrentGear          : WORD := 523;(*Transmission Current Gear*)

(*Transmission Control 1 - TC1*)
	wPGN_TC1                             : WORD := 256;
	tRPT_TC1                             : TIME := T#0ms;(*Transmission Repetition Rate*)
	byLEN_TC1                            : BYTE := 8;(*Data Length (Number of bytes to be transmitted)*)
	byPG_TC1                             : BYTE := 0;(*Data Page (Page address)*)
	byPDUFormat_TC1                      : BYTE := 1;
	byPDUSpecific_TC1                    : BYTE := 3;(*DA, 3 или 6 - ?;*)
	byPRIO_TC1                           : BYTE := 3;(*Default Priority (Message priority)*)

	SPN_RequestedGear                    : WORD := 525;(*Requested Gear*)

(*ACTIVE DIAGNOSTIC TROUBLE CODES - DM1*)
	wPGN_DM1                             : WORD := 65226;(*16#00FECA00*)
	tRPT_DM1                             : TIME := T#0S;(*Transmission Repetition Rate, variable*)
	byLEN_DM1                            : BYTE := 8;(*Data Length (Number of bytes to be transmitted)*)
	byPG_DM1                             : BYTE := 0;(*Data Page (Page address)*)
	byPDUFormat_DM1                      : BYTE := 254;
	byPDUSpecific_DM1                    : BYTE := 202;
	byPRIO_DM1                           : BYTE := 6;(*Default Priority (Message priority)*)

(*PREVIOUSLY ACTIVE DIAGNOSTIC TROUBLE CODES - DM2*)
	wPGN_DM2                             : WORD := 65227;(*16#00FECB00*)
	tRPT_DM2                             : TIME := T#0s;(*Transmission Repetition Rate, variable*)
	byLEN_DM2                            : BYTE := 8;(*Data Length (Number of bytes to be transmitted)*)
	byPG_DM2                             : BYTE := 0;(*Data Page (Page address)*)
	byPDUFormat_DM2                      : BYTE := 254;
	byPDUSpecific_DM2                    : BYTE := 203;
	byPRIO_DM2                           : BYTE := 6;(*Default Priority (Message priority)*)

(*Torque/Speed Control 1 - TSC1*)
	wPGN_TSC1                             : WORD := 0;(*16#00000000*)
	tRPT_TSC1                             : TIME := T#10ms;(*Transmission Repetition Rate*)
	byLEN_TSC1                            : BYTE := 8;(*Data Length (Number of bytes to be transmitted)*)
	byPG_TSC1                             : BYTE := 0;(*Data Page (Page address)*)
	byPDUFormat_TSC1                      : BYTE := 0;
	byPDUSpecific_TSC1                    : BYTE := 16#DA;(*DA, 3 или 6 - ?;*)
	byPRIO_TSC1                           : BYTE := 3;(*Default Priority (Message priority)*)

	SPN_RequestedSpeed_SpeedLimit         : WORD := 898;(*Requested Speed/Speed Limit*)

(*Cruise Control/Vehicle Speed - CCVS*)
	wPGN_CCVS                             : WORD := 65265;(*16#00FEF100*)
	tRPT_CCVS                             : TIME := T#100ms;(*Transmission Repetition Rate*)
	byLEN_CCVS                            : BYTE := 8;(*Data Length (Number of bytes to be transmitted)*)
	byPG_CCVS                             : BYTE := 0;(*Data Page (Page address)*)
	byPDUFormat_CCVS                      : BYTE := 254;
	byPDUSpecific_CCVS                    : BYTE := 241;(*DA, 3 или 6 - ?;*)
	byPRIO_CCVS                           : BYTE := 6;(*Default Priority (Message priority)*)

	SPN_ParkingBrakeSwitch                : WORD := 70;(*Parking Brake Switch*)
	SPN_WheelBasedVehicleSpeed            : WORD := 84;(*Wheel-Based Vehicle Speed*)
	SPN_CruiseControlEnableSwitch         : WORD := 596;(*Cruise Control Enable Switch*)
	SPN_BrakeSwitch                       : WORD := 597;(*Brake Switch*)
	SPN_ClutchSwitch                      : WORD := 598;(*Clutch Switch*)
	SPN_CruiseControlSetSwitch            : WORD := 599;(*Cruise Control Set Switch*)
	SPN_CruiseControlDecelerateSwitch     : WORD := 600;(*Cruise Control Coast (Decelerate) Switch*)
	SPN_CruiseControlResumeSwitch         : WORD := 601;(*Cruise Control Resume Switch*)
	SPN_CruiseControlAccelerateSwitch     : WORD := 602;(*Cruise Control Accelerate Switch*)
END_VAR

(* Global variable list: GV_Control *)
VAR_GLOBAL
(*Управление процессом 1*)
	byRequestNextStep              : BYTE := 0 ;(* =REQ_STAGE:BYTE; 0x0003  Запрос перехода на следующий этап*)
	W_REQ_STAGE                    : BYTE; (*0x0003  Запрос перехода на следующий этап, для панели ?, запись*)
	R_REQ_STAGE                    : BYTE; (*0x0003  Запрос перехода на следующий этап, для панели ?, чтение*)

	bControlExecutionSteps         : ARRAY[1..7] OF BOOL; (*Контроль выполнения шагов*)
    byCurrentSubStep               : BYTE := 0; (*Tекущий субшаг, == 0 если шаг не имеет подшага*)

												  (*Kод ошибки шага
	 												= 0 - нет ошибки
	 												= номеру задаваемого шага - предыдущий шаг не выполнен*)
	byErrorStepPC                  : BYTE := 0;  (*Kод ошибки для PC*)
    byErrorStepPan                 : BYTE := 0;  (*Kод ошибки для панели*)
	dwErrorConditionRunStep        : DWORD := 0; (*NOT 0 - не сформированы условия необходимые для выполнения*)

	wCurrentStageOperation         : WORD;(*0x0030 Текущий этап алгоритма:
													- 0 байт - текущий шаг;
													- 1 байт - теущий суб-шаг*)

	byStageCondition               : BYTE; (*0x0031 - Состояние шага:
													- 0 - работает;
													- 1 - останов по ошибке;
													- 2 - работает с ошибкой;
													- 3 - окончен*)

	diRequiredStageOperation       : DINT  := 0;(*Требуемый этап работы*)
	byCurrStep                     : BYTE  := 0;(*Tекущий этап*)

(*Управление процессом 2*)
	bDefaultSettings               : BOOL  := 0;(*Команда 01*)  (*"Сброс установок в заводские значения"*)
	bStart                         : BOOL  := 0;                (*Состояние кнопки "Старт"/"Стоп"*)
	bStop                          : BOOL  := 0;(*Команда 02*)  (*"Стоп"*)
	dwProcessState                 : DWORD := 0;                (*Состояние процесса*)
	bHornDisable                   : BOOL  := 0;(*Команда 03*)  (*"Запретить работу звукового сигнала"*)
	dwHornEnable                   : DWORD := 0;                (*Разрешение работы звукового сигнала*)
	bBlockDisable                  : BOOL  := 0;(*Команда 04*)  (*"Отключение блокировки"*)
	bResetTotalAmountGN2           : BOOL  := 0;                (*Обнуление общего объема закачанного азота*)
	bPressSensorRST                : BOOL  := 0;                (*"Обнулить датчик давления нагнетания"*)
	byAutoModeDisplay              : BYTE  := 1;(*Режим работы контроллера, задаваемый с дисплея, "Авто"/"Ручное", 1 - "Авто", 0 - "Ручное"*)

(*Управление двигателем*)
	diRequiredEngineRPM            : DINT  :=   0 (*750*);(*Требуемые обороты двигателя*)
	diCurrentEngineRPM             : DINT  :=   0;(*Текущие обороты двигателя*)
	diRecommendEngineRPM           : DINT  :=   0;(*Рекомендуемые обороты двигателя*)
	diIdlingEngineRPM              : DINT  := 750;(*Обороты холостого хода двигателя*)

	diRequiredNumberGear           : DINT  := 0;(*Требуемая передача АКПП*)
	diCurrentNumberGear            : DINT  := 0;(*Текущая передача АКПП*)
	diRecommendNumberGear          : DINT  := 0;(*Рекомендуемая передача АКПП*)

	byTorqueConverterLockupEngaged : BYTE  := 0;(**)
END_VAR

(* Global variable list: GV_Errors *)
VAR_GLOBAL
(*Ошибки по аналоговым входам*)
	bErrorBoostPres       : BOOL := 0;(*Флаг ошибки аналогового канала 1*)
	bErrorLN2_Temp        : BOOL := 0;(*Флаг ошибки аналогового канала 2*)

	bErrorGN2_Temp        : BOOL := 0;(*Флаг ошибки аналогового канала 4*)
	bErrorGN2_Pres        : BOOL := 0;(*Флаг ошибки аналогового канала 5*)
	bErrorHydHeatPres     : BOOL := 0;(*Флаг ошибки аналогового канала 6*)
	bErrorSpare01         : BOOL := 0;(*Флаг ошибки аналогового канала 7*)
	bErrorSpare02         : BOOL := 0;(*Флаг ошибки аналогового канала 8*)

	bErrorCoolTempIn      : BOOL := 0;(*Флаг ошибки аналогового канала 9*)
	bErrorSpare03         : BOOL := 0;(*Флаг ошибки аналогового канала 10*)

	bErrorSpare04         : BOOL := 0;(*Флаг ошибки аналогового канала 12*)

	bErrorSpare05         : BOOL := 0;(*Флаг ошибки аналогового канала 14*)
	bErrorSpare06         : BOOL := 0;(*Флаг ошибки аналогового канала 15*)
	bErrorSpare07         : BOOL := 0;(*Флаг ошибки аналогового канала 16*)

	bCommomErrorADC       : BOOL := 0;

	bArrayErrorADC        : ARRAY [1..32] OF BOOL;(*Состояния каналов по обрывам и КЗ*)

	dwErrorADC_MS         : DWORD := 0;
	dwErrorADC_SL1        : DWORD := 0;
	dwErrorADC_SL2        : DWORD := 0;
	dwErrorADC_SL3        : DWORD := 0;

(*Ошибки*)
	bErrorNumber01        : BOOL := 0;(*Ошибка 01. Нет связи с компьютерной панелью,                                                       РАБОТАЕМ С ПРЕДУПРЕЖДЕНИЕМ*)
	bErrorNumber02        : BOOL := 0;(*Ошибка 02. Температура газообразного азота ниже допустимого аварийного уровня,                     РАБОТАЕМ С ПРЕДУПРЕЖДЕНИЕМ*)
	bErrorNumber03        : BOOL := 0;(*Ошибка 03. Температура газообразного азота выше допустимого аварийного уровня,                     РАБОТАЕМ С ПРЕДУПРЕЖДЕНИЕМ*)
	bErrorNumber04        : BOOL := 0;(*Ошибка 04. Превышение давление газообразного азота,                                                ОСТАНОВ НВД*)
	bErrorNumber05        : BOOL := 0;(*Ошибка 05. Аварийный останов двигателя,                                                            ОСТАНОВ И УХОДИМ НА НАЧАЛО*)
	bErrorNumber06        : BOOL := 0;(*Ошибка 06. Обороты двигателя 0,                                                                    ОСТАНОВ И УХОДИМ НА НАЧАЛО*)
	bErrorNumber07        : BOOL := 0;(*Ошибка 07. Блокировка НВД отключена. Максимум 20 об.мин,                                           РАБОТАЕМ С ПРЕДУПРЕЖДЕНИЕМ*)
	bErrorNumber08        : BOOL := 0;(*Ошибка 08. Ошибка CAN2 J1939,                                                                      РАБОТАЕМ С ПРЕДУПРЕЖДЕНИЕМ*)
	bErrorNumber09        : BOOL := 0;(*Ошибка 09. Отсутсвует CAN2 J1939,                                                                  ОСТАНОВ И УХОДИМ НА НАЧАЛО*)
	bErrorNumber10        : BOOL := 0;(*Ошибка 10. Тумблер управления подкачивающим насосом перевести в "Ручной",                          РАБОТАЕМ С ПРЕДУПРЕЖДЕНИЕМ. ИНИЦИАЛИЗАЦИЯ*)
	bErrorNumber11        : BOOL := 0;(*Ошибка 11. Тумблер НВД перевести в "Ручной",                                                       РАБОТАЕМ С ПРЕДУПРЕЖДЕНИЕМ. ИНИЦИАЛИЗАЦИЯ*)
	bErrorNumber12        : BOOL := 0;(*Ошибка 12. Тумблер управления гидронагрева перевести в "Ручной",                                   РАБОТАЕМ С ПРЕДУПРЕЖДЕНИЕМ. ИНИЦИАЛИЗАЦИЯ*)
	bErrorNumber13        : BOOL := 0;(*Ошибка 13. НВД. Температура жидкого азота выше допустимого уровня,                                 ОСТАНОВ НВД (-> + ОСТАНОВ ГИДРОНАГРЕВА)*)
	bErrorNumber14        : BOOL := 0;(*Ошибка 14. НВД. Давление подпитки ниже допустимого уровня,                                         ОСТАНОВ НВД (-> + ОСТАНОВ ГИДРОНАГРЕВА)*)
	bErrorNumber15        : BOOL := 0;(*Ошибка 15. НВД. Температура ОЖ теплобменника ниже допустимого уровня,                              ОСТАНОВ НВД (-> + ОСТАНОВ ГИДРОНАГРЕВА)*)
	bErrorNumber16        : BOOL := 0;(*Ошибка 16. НВД. Проверьте ручное управление,                                                       РАБОТАЕМ С ПРЕДУПРЕЖДЕНИЕМ*)

	bErrorNumber17        : BOOL := 0;(*Ошибка 17. Подкачивающий насос. Температура жидкого азота выше допустимого уровня,                 ОСТАНОВ ПОДКАЧИВАЮЩЕГО НАСОСА*)
	bErrorNumber18        : BOOL := 0;(*Ошибка 18. Подкачивающий насос. Проверьте ручное управление,                                       РАБОТАЕМ С ПРЕДУПРЕЖДЕНИЕМ*)
	bErrorNumber19        : BOOL := 0;(*Ошибка 19. Гидронагрев. Температура жидкого азота выше допустимого уровня,                         ОСТАНОВ ГИДРОНАГРЕВА*)
	bErrorNumber20        : BOOL := 0;(*Ошибка 20. Гидронагрев. Давление подпитки ниже допустимого уровня,                                 ОСТАНОВ ГИДРОНАГРЕВА*)
	bErrorNumber21        : BOOL := 0;(*Ошибка 21. Гидронагрев. Температура ОЖ теплобменника ниже допустимого уровня,                      ОСТАНОВ ГИДРОНАГРЕВА*)
	bErrorNumber22        : BOOL := 0;(*Ошибка 22. Гидронагрев. Скорость НВД меньше 20 об/мин,                                             ОСТАНОВ ГИДРОНАГРЕВА*)
	bErrorNumber23        : BOOL := 0;(*Ошибка 23. Гидронагрев. Проверьте ручное управление,                                               РАБОТАЕМ С ПРЕДУПРЕЖДЕНИЕМ*)
	bErrorNumber24        : BOOL := 0;(*Ошибка 24. Проверьте состояние органов ручного управления                                          РАБОТАЕМ С ПРЕДУПРЕЖДЕНИЕМ*)
	bErrorNumber25        : BOOL := 0;(*Ошибка 25. *)
	bErrorNumber26        : BOOL := 0;(*Ошибка 26. *)
	bErrorNumber27        : BOOL := 0;(*Ошибка 27. *)
	bErrorNumber28        : BOOL := 0;(*Ошибка 28. *)
	bErrorNumber29        : BOOL := 0;(*Ошибка 29. *)
	bErrorNumber30        : BOOL := 0;(*Ошибка 30. *)
	bErrorNumber31        : BOOL := 0;(*Ошибка 31. *)
	bErrorNumber32        : BOOL := 0;(*Ошибка 32. *)

	dwErrorState          : DWORD := 0;(*Состояние ошибок, сообщения*)
	bResetErrors          : BOOL  := 0;(*Сброс ошибок*)
END_VAR

(* Global variable list: GV_FRAM *)
VAR_GLOBAL
END_VAR

VAR_GLOBAL CONSTANT
(*Установка начальных адресов для блоков данных массива параметров каналов, считаем по 256 байт на каждый блок (64 * DWORD)*)
	iMemAdrArrayParam00        : INT :=    0;(*Начальный адрес блока параметров 00 в энергонезависимой памяти*)
	iMemAdrArrayParam01        : INT :=  256;(*Начальный адрес блока параметров 01 в энергонезависимой памяти*)
	iMemAdrArrayParam02        : INT :=  512;(*Начальный адрес блока параметров 02 в энергонезависимой памяти*)
	iMemAdrArrayParam03        : INT :=  768;(*Начальный адрес блока параметров 03 в энергонезависимой памяти*)
	iMemAdrArrayParam04        : INT := 1024;(*Начальный адрес блока параметров 04 в энергонезависимой памяти*)
	iMemAdrArrayParam05        : INT := 1280;(*Начальный адрес блока параметров 05 в энергонезависимой памяти*)
	iMemAdrArrayParam06        : INT := 1536;(*Начальный адрес блока параметров 06 в энергонезависимой памяти*)
	iMemAdrArrayParam07        : INT := 1792;(*Начальный адрес блока параметров 07 в энергонезависимой памяти*)
	iMemAdrArrayParam08        : INT := 2048;(*Начальный адрес блока параметров 08 в энергонезависимой памяти*)
	iMemAdrArrayParam09        : INT := 2304;(*Начальный адрес блока параметров 09 в энергонезависимой памяти*)
	iMemAdrArrayParam10        : INT := 2560;(*Начальный адрес блока параметров 10 в энергонезависимой памяти*)

(*Установка начальных адреса для блока имен параметров каналов, считаем по 2048 байт на блок (64 * 8 * DWORD)*)
	iMemAdrArrayParamName      : INT := 2816;(*Начальный адрес блока параметров Name в энергонезависимой памяти*)

(*Сервисные значения*)
	iMemAdrFirstStartId        : INT := 5000;(**)
	iMemAdrTotalServiceMeter   : INT := 5010;(*Адрес сохранения моточасов в энергонезависимой памяти*)
	iMemAdrCurrCANAddr         : INT := 5020;(*Адрес сохранения текущего адреса на шине CAN PC в энергонезависимой памяти*)
	iMemAdrCurrMode            : INT := 5030;(*Адрес сохранения текущего режима работы установки в энергонезависимой памяти*)
	iMemAdrCHANNEL_INDEX       : INT := 5040;(*Адрес сохранения индекса текущего канала*)

(*Технологические установки*)
	iMemAdrSet_GN2TempManual   : INT := 5110;(**)
	iMemAdrSet_GN2OverPres     : INT := 5120;(**)
	iMemAdrSet_BoostPresManual : INT := 5130;(**)
	iMemAdrSet_GN2Rate         : INT := 5140;(**)
	iMemAdrSet_LN2SaturTemp    : INT := 5150;(**)

	iMemAdrPINAdder            : ARRAY [0..7] OF INT := 5200, 5210, 5220, 5230, 5240, 5250, 5260, 5270;(*Адреса расходомеров в энергонезависимой памяти*)
END_VAR

(* Global variable list: GV_IO *)
VAR_GLOBAL
(*Переменные аналоговых каналов*)
	rArrayDataRAWADC         : ARRAY [1..16] OF REAL;(*Массив необработанных неусредненных данных каналов*)
	rADC_ValueHigh           : REAL  := 3430;
	rADC_ValueLow            : REAL  := 588;

(*Переменные частотных каналов*)
	rArrayDataRAWPIN         : ARRAY [1..8] OF REAL;(*Массив необработанных данных каналов*)
	rFRQ_ValueHigh           : REAL  := 50_000;
	rFRQ_ValueLow            : REAL  := -1;

(*Переменные каналов ШИМ*)
	rArrayDataRAWPWM         : ARRAY [1..8] OF REAL;(*Массив необработанных данных каналов*)

(*Переменные каналов ПИД*)
	rArrayDataRAWPID         : ARRAY [1..8] OF REAL;(*Массив необработанных данных каналов*)

(*Переменные сумматоров частотных входов*)
	udiArrayDataPINAdderOut   : ARRAY [1..8] OF UDINT;(*Массив выходных значений суммирующих каналов*)
	bArrayDataPINAdderReset   : ARRAY [1..8] OF BOOL;(*Массив флагов сброса выходных значений суммирующих каналов*)

	bFlowmeterReset_1         : BOOL;(*Флаг сброса сумматора частотного канала 0*)
	bFlowmeterReset_2         : BOOL;(*Флаг сброса сумматора частотного канала 1*)
	bFlowmeterReset_3         : BOOL;(*Флаг сброса сумматора частотного канала 2*)
	bFlowmeterReset_4         : BOOL;(*Флаг сброса сумматора частотного канала 3*)

(*Дискретные входы*)
	bIX_TriplexRPMAutoMode    : BOOL := 0;(*Авто/Ручной режим рег. оборотов НВД*)
	bIX_HydHeatPresAutoMode   : BOOL := 0;(*Авто/Ручной режим рег. гидронагрева*)
	bIX_BoostPresAutoMode     : BOOL := 0;(*Авто/Ручной режим рег. центробежного насоса*)
	bIX_BlockOff              : BOOL := 0;(*Отключение блокировки*)
	bIX_EngineStopped         : BOOL := 0;(*Аварийная остановка двигателя Detroit*)

	IX_Test                   : BOOL := 0;(*Тест ламп*)

	dwInputState              : DWORD := 0;

(*Выходы ПИД*)
	rPID_HydHeatPres          : REAL := 0;(*Регулировка давления гидронагрева*)
	rPID_TriplexRPM           : REAL := 0;(*Регулировка оборотов НВД*)
	rPID_BoostPres            : REAL := 0;(*Регулировка давления центробежного насоса*)

(*Выходы ШИМ*)
	rPWM_HydHeatPres          : REAL := 0;(*Регулировка давления гидронагрева*)
	rPWM_TriplexRPM           : REAL := 0;(*Регулировка оборотов НВД*)
	rPWM_BoostPres            : REAL := 0;(*Регулировка давления центробежного насоса*)

(*Дискретные выходы*)
	bQX_TriplexEmergStop      : BOOL := 0;(*Аварийная остановка НВД*)
	bQX_TriplexEmergStopTrig  : BOOL := 0;(*Аварийная остановка НВД (с триггером)*)

	bQX_Horn                  : BOOL := 0;(*Звуковой сигнал*)
	bQX_EngineStarterBlock    : BOOL := 0;(*Блокировка запуска двигателя*)
	bQX_TriplexRPMContrMode   : BOOL := 0;(*Режим рег. оборотов НВД*)
	bQX_HydHeatPresContrMode  : BOOL := 0;(*Режим рег. гидронагрева*)
	bQX_BoostPresContrMode    : BOOL := 0;(*Режим рег. давления центробежного насоса*)

	dwOutputState             : DWORD := 0;
END_VAR

(* Global variable list: GV_Parameters *)
VAR_GLOBAL
(*Параметры аналоговых входов*)
	rIW_GN2_Temp              : REAL := 0;(*Температура нагнетания*)
	rIW_GN2_Pres              : REAL := 0;(*Давление нагнетания*)
	rIW_LN2_Temp              : REAL := 0;(*Температура азота жидкого*)
	rIW_BoostPres             : REAL := 0;(*Давление подпитки*)
	rIW_HydHeatPres           : REAL := 0;(*Давление гидронагрева*)
	rIW_CoolTempIn            : REAL := 0;(*Температура ОЖ до испарителя*)

	rWF_PresCor              : REAL := 0;(*Корректировка давления нагнетания*)
	rWF_PresOut              : REAL := 0;(*Корректированное давление нагнетания*)

(*Параметры частотные входов*)
	rFRQ_TriplexRPM           : REAL := 0;(*Обороты НВД*)

(*Параметры процесса*)
	rCurrent_GN2Rate         : REAL :=   0;(*Текущая производительность установки, м3/мин*)
	udiCurrent_GN2RateLitres : UDINT :=   0;(*Текущая производительность установки, л3/мин*)
	rTotalAmountGN2          : REAL :=   0;(*Общий объем закачанного азота, м3*)
	rTotalAmountGN2NotReset  : REAL :=   0;(*Общий объем закачанного азота (несбрасываемый), м3*)

(*Установки процесса*)
	rSet_GN2Rate             : REAL :=   0;(*Требуемая производительность установки*)
	rSetTotalAmountGN2       : REAL := 100;(*Требуемый общий объем закачанного азота, м3*)
	rSet_LN2SaturTemp        : REAL :=-170;(*Температура азота, когда можно переходить к управлению подкачивающим насосом, С (задается с КП !!!)*)
	rSet_LN2SaturTempTriplex : REAL :=-181;(*Температура азота, когда можно переходить к управлению НВД и гидронагревом, С (с КП НЕ задается !!!)*)
	rSet_GN2OverPres         : REAL :=  70;(*Установка предельно-допустимого давления газообразного азота, МПа*)

	bHydHeatPresMode         : BOOL :=   0;(*Управление давлением гидронагрева "Авто"/"Ручное"*)
	rSet_GN2Temp             : REAL :=   0;(*Установка температуры (текущая) гидронагрева, авто/корректировка*)
	rSet_GN2TempAuto         : REAL :=   0;(*Установка температуры гидронагрева в автоматическом режиме*)
	rSet_GN2TempManual       : REAL :=   0;(*Установка ручной корректировки температуры гидронагрева*)
	bHydHeatPresEnable       : BOOL :=   0;(*Разрешение работы гидронагрева*)
	bHydHeatPresDisparity    : BOOL :=   0;(**)
	bSet_HydHeatPresManual   : BOOL :=   0;(*Признак ручной корректировки давления гидронагрева*)
	rHydHeatPres_Err         : REAL :=   0;(**)
	rHydHeatPres_Calc        : REAL :=   0;(**)

	bTriplexRPMMode          : BOOL :=   0;(*Управление скоростью НВД "Авто"/"Ручное"*)
	rSet_TriplexRPM          : REAL :=   0;(*Установка скорости (текущая) НВД, авто/корректировка*)
	rSet_TriplexRPMAuto      : REAL :=   0;(*Установка скорости НВД в автоматическом режиме*)
	rSet_TriplexRPMManual    : REAL :=   0;(*Установка ручной корректировки скорости НВД*)
	bTriplexRPMEnable        : BOOL :=   0;(*Разрешение работы НВД*)
	bTriplexRPMDisparity     : BOOL :=   0;(**)
	bSet_TriplexRPMManual    : BOOL :=   0;(*Признак ручной корректировки скорости НВД*)

	rCoolTempInMin           : REAL :=   0;(*Минимальная температура ОЖ до испарителя*)
	rTriplexRPM_Err          : REAL :=   0;(**)
	rTriplexRPM_Calc         : REAL :=   0;(**)

	bBoostPresMode           : BOOL :=   0;(*Управление давлением подпитки "Авто"/"Ручное"*)
	rSet_BoostPres           : REAL :=   0;(*Установка давления (текущая) подпитки, авто/корректировка*)
	rSet_BoostPresAuto       : REAL := 0.6;(*Установка давления подпитки в автоматическом режиме*)
	rSet_BoostPresManual     : REAL := 0.6;(*Установка ручной корректировки давления подпитки*)
	bBoostPresEnable         : BOOL :=   0;(*Разрешение работы насоса подпитки(подкачки)*)
	bBoostPresDisparity      : BOOL :=   0;(**)
	bSet_BoostPresManual     : BOOL :=   0;(*Признак ручной корректировки давления подпитки*)
END_VAR

(* Global variable list: GV_Service *)
VAR_GLOBAL
(*Идентификатор программы*)
	abyMS_ProgramID         : ARRAY [0..3] OF BYTE;

	byProgrammableDeviceType     : BYTE  := 16#0; (*Тип программируемого прибора*)
	byUnitTypePrimaryApp         : BYTE  := 16#4; (*Тип установки первичного применения*)
	byUnitModelPrimaryApp        : BYTE  := 16#2; (*Модель установки первичного применения*)
	byUnitModificationPrimaryApp : BYTE  := 16#2; (*Модификация установки первичного применения*)
	byFixNumber                  : BYTE  := 16#1;(*Номер исправления*)

	dwMS_ProgramCRC         : DWORD := 0;

(*Системное время*)
	dwTime_US               : DWORD := 10;
	dwCycleTime             : DWORD := 0;

(*Сигнал управления морганием лампочек*)
	bTimerBlinkOut          : BOOL  := 0;

(*Состояние системы*)
	abyDataStateMS          : ARRAY [0..3] OF BYTE;
	abyDataStateSL1         : ARRAY [0..3] OF BYTE;
	abyDataStateSL2         : ARRAY [0..3] OF BYTE;
	abyDataStateSL3         : ARRAY [0..3] OF BYTE;

(*Напряжения питания контроллеров в сети*)
	rECU_SupplyVoltage      : REAL := 0;

(*Температура контроллеров в сети*)
	rECU_Temperature        : REAL := 0;

(*Время наработки*)
	rTotalServiceMeterOut   : REAL;(*Суммарно наработанные моточасы, на отправку*)
	rLastServiceMeterOut    : REAL:=0;(*Наработанные моточасы с последнего включения, на отправку*)

	dwTotalServiceMeter     : DWORD;(*Суммарно наработанные моточасы*)
	dwLastServiceMeter      : DWORD := 0;(*Наработанные моточасы с последнего включения*)

	byButtonPowerStatus     : BYTE := 0;
END_VAR

(* Data type *)
TYPE CAN1_ERROR_DM1 :
	STRUCT
		dwSPN       : DWORD;
		byFMI       : BYTE;
		byOC        : BYTE;
		byErrorsQty : BYTE;
		byLampState : BYTE;
	END_STRUCT
END_TYPE

(* Data type *)
TYPE CAN1_ERROR_DM2 :
	STRUCT
		dwSPN       : DWORD;
		byFMI       : BYTE;
		byOC        : BYTE;
		byErrorsQty : BYTE;
		byLampState : BYTE;
	END_STRUCT
END_TYPE

(* Data type *)
TYPE Page_Channel :
	STRUCT
		PARAM_NAME : STRING(32);
		PARAM_00   : DWORD;
		PARAM_01   : REAL;
		PARAM_02   : REAL;
		PARAM_03   : REAL;
		PARAM_04   : REAL;
	    PARAM_05   : DWORD;
		PARAM_06   : REAL;
		PARAM_07   : DWORD;
		PARAM_08   : REAL;
		PARAM_09   : DWORD;
        PARAM_10   : REAL;
	END_STRUCT
END_TYPE

(* POU PLC_PRG, FBD *)
PROGRAM PLC_PRG

VAR
	init_1        : BOOL := TRUE;
	init_e        : BOOL;
	cycletime     : DWORD;
	max_cycletime : DWORD;
	reset_max     : BOOL;
END_VAR
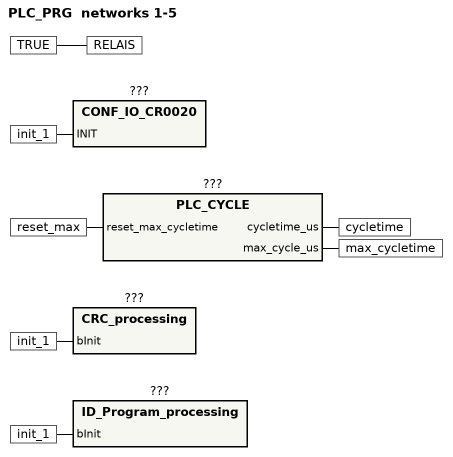
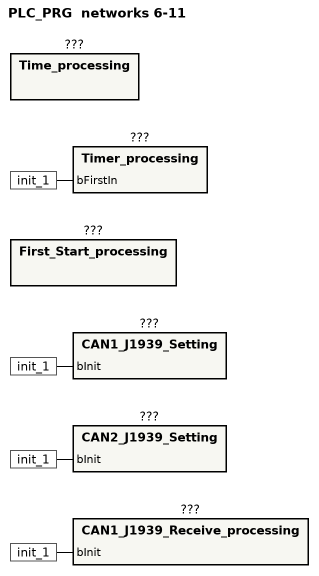
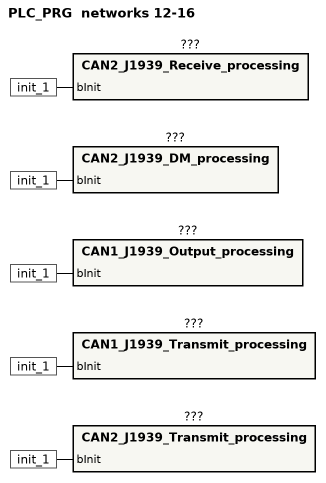
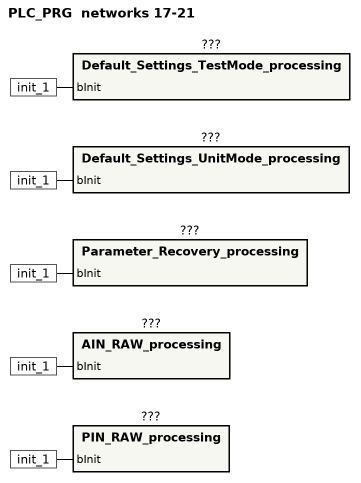
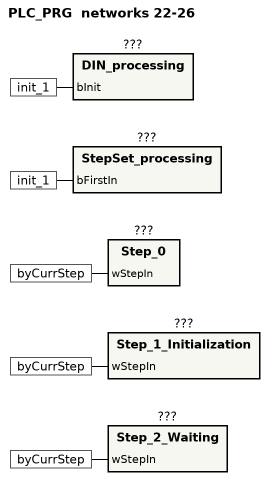
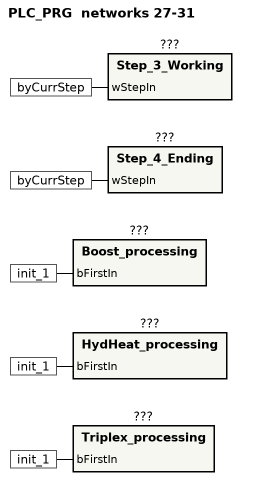
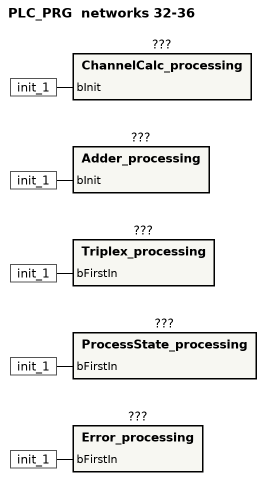
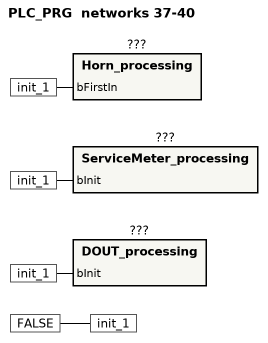
_FBD_ (* Function Block Diagram *)
NETWORK 1
	TRUE => RELAIS
NETWORK 2
	???:CONF_IO_CR0020(INIT: init_1)
NETWORK 3 (* For monitoring *)
	???:PLC_CYCLE(reset_max_cycletime: reset_max, max_cycle_us => max_cycletime) => cycletime
NETWORK 4
	???:CRC_processing(bInit: init_1)
NETWORK 5
	???:ID_Program_processing(bInit: init_1)
NETWORK 6
	???:Time_processing()
NETWORK 7
	???:Timer_processing(bFirstIn: init_1)
NETWORK 8
	???:First_Start_processing()
NETWORK 9
	???:CAN1_J1939_Setting(bInit: init_1)
NETWORK 10
	???:CAN2_J1939_Setting(bInit: init_1)
NETWORK 11
	???:CAN1_J1939_Receive_processing(bInit: init_1)
NETWORK 12
	???:CAN2_J1939_Receive_processing(bInit: init_1)
NETWORK 13
	???:CAN2_J1939_DM_processing(bInit: init_1)
NETWORK 14
	???:CAN1_J1939_Output_processing(bInit: init_1)
NETWORK 15
	???:CAN1_J1939_Transmit_processing(bInit: init_1)
NETWORK 16
	???:CAN2_J1939_Transmit_processing(bInit: init_1)
NETWORK 17
	???:Default_Settings_TestMode_processing(bInit: init_1)
NETWORK 18
	???:Default_Settings_UnitMode_processing(bInit: init_1)
NETWORK 19
	???:Parameter_Recovery_processing(bInit: init_1)
NETWORK 20
	???:AIN_RAW_processing(bInit: init_1)
NETWORK 21
	???:PIN_RAW_processing(bInit: init_1)
NETWORK 22
	???:DIN_processing(bInit: init_1)
NETWORK 23
	???:StepSet_processing(bFirstIn: init_1)
NETWORK 24
	???:Step_0(wStepIn: byCurrStep)
NETWORK 25
	???:Step_1_Initialization(wStepIn: byCurrStep)
NETWORK 26
	???:Step_2_Waiting(wStepIn: byCurrStep)
NETWORK 27
	???:Step_3_Working(wStepIn: byCurrStep)
NETWORK 28
	???:Step_4_Ending(wStepIn: byCurrStep)
NETWORK 29
	???:Boost_processing(bFirstIn: init_1)
NETWORK 30
	???:HydHeat_processing(bFirstIn: init_1)
NETWORK 31
	???:Triplex_processing(bFirstIn: init_1)
NETWORK 32
	???:ChannelCalc_processing(bInit: init_1)
NETWORK 33
	???:Adder_processing(bInit: init_1)
NETWORK 34
	???:Triplex_processing(bFirstIn: init_1)
NETWORK 35
	???:ProcessState_processing(bFirstIn: init_1)
NETWORK 36
	???:Error_processing(bFirstIn: init_1)
NETWORK 37
	???:Horn_processing(bFirstIn: init_1)
NETWORK 38
	???:ServiceMeter_processing(bInit: init_1)
NETWORK 39
	???:DOUT_processing(bInit: init_1)
NETWORK 40 (* Last line *)
	FALSE => init_1
_END_FBD_
(* the same logic as Structured Text *)
(* Network 1 *)
RELAIS := TRUE;
(* Network 2: see the listing above *)
(* Network 3: see the listing above *)
(* Network 4: see the listing above *)
(* Network 5: see the listing above *)
(* Network 6: see the listing above *)
(* Network 7: see the listing above *)
(* Network 8: see the listing above *)
(* Network 9: see the listing above *)
(* Network 10: see the listing above *)
(* Network 11: see the listing above *)
(* Network 12: see the listing above *)
(* Network 13: see the listing above *)
(* Network 14: see the listing above *)
(* Network 15: see the listing above *)
(* Network 16: see the listing above *)
(* Network 17: see the listing above *)
(* Network 18: see the listing above *)
(* Network 19: see the listing above *)
(* Network 20: see the listing above *)
(* Network 21: see the listing above *)
(* Network 22: see the listing above *)
(* Network 23: see the listing above *)
(* Network 24: see the listing above *)
(* Network 25: see the listing above *)
(* Network 26: see the listing above *)
(* Network 27: see the listing above *)
(* Network 28: see the listing above *)
(* Network 29: see the listing above *)
(* Network 30: see the listing above *)
(* Network 31: see the listing above *)
(* Network 32: see the listing above *)
(* Network 33: see the listing above *)
(* Network 34: see the listing above *)
(* Network 35: see the listing above *)
(* Network 36: see the listing above *)
(* Network 37: see the listing above *)
(* Network 38: see the listing above *)
(* Network 39: see the listing above *)
(* Network 40 *)
init_1 := FALSE;
END_PROGRAM

(* POU I_O_CONFIGURATION/CONF_IO_CR0020, FBD *)
PROGRAM CONF_IO_CR0020

VAR CONSTANT
	(*IN_NOMODE ==> all Bits 0*)
	IN_DIGITAL_H_            : BOOL := TRUE;(*Bit 0*)
	IN_DIGITAL_L_            : BOOL := TRUE;(*Bit 1*)
	IN_CURRENT_              : BOOL := TRUE;(*Bit 2*)
	IN_VOLTAGE10_            : BOOL := TRUE;(*Bit 3*)
	IN_VOLTAGE30_            : BOOL := TRUE;(*Bit 4*)
	IN_RATIO_                : BOOL := TRUE;(*Bit 5*)
	IN_DIAGNOSTIC_           : BOOL := TRUE;(*Bit 6*)
	IN_FAST_                 : BOOL := TRUE;(*Bit 7*)

	(*OUT_NOMODE ==> all bits 0*)
	OUT_DIGITAL_H_           : BOOL := TRUE;(*Bit 0*)
	OUT_DIGITAL_L_           : BOOL := TRUE;(*Bit 1*)
	OUT_CURRENT_             : BOOL := TRUE;(*Bit 2*)

	OUT_DIAGNOSTIC_          : BOOL := TRUE;(*Bit 6*)
	OUT_OVERLOAD_PROTECTION_ : BOOL := TRUE;(*Bit 7*)
END_VAR

VAR_INPUT
	INIT: BOOL;
END_VAR
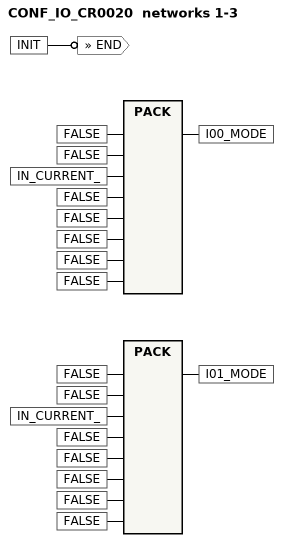
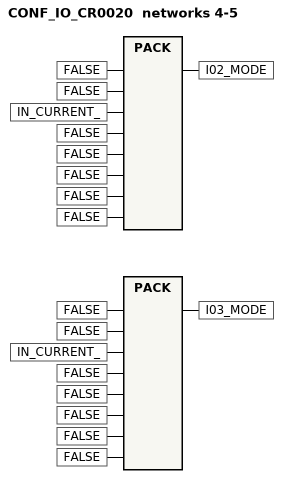
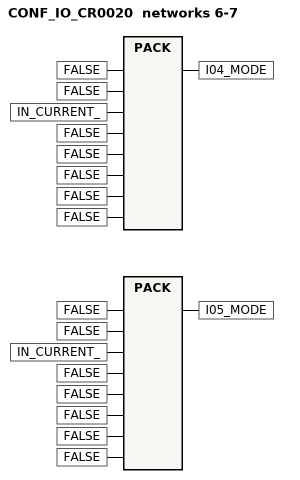
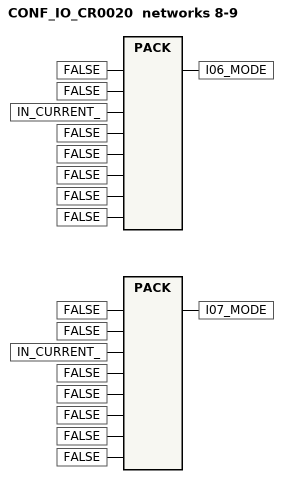
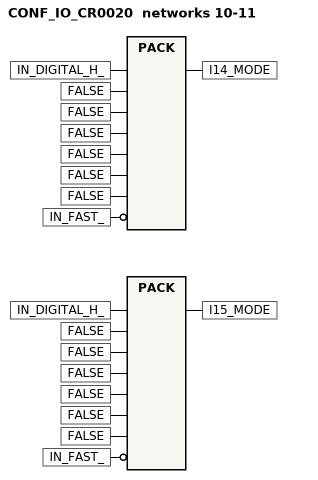
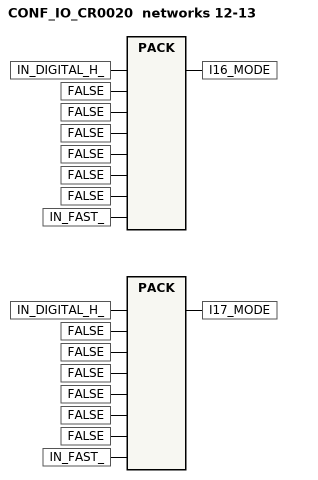
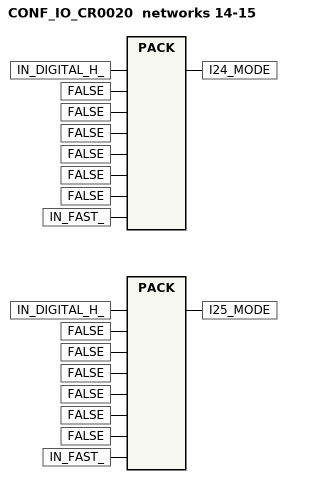
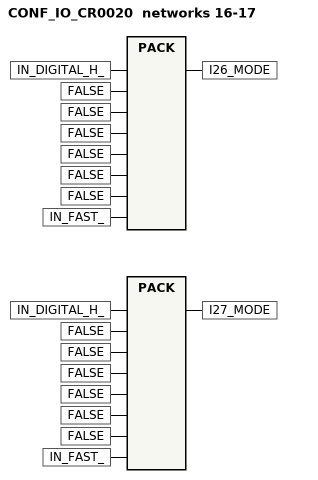
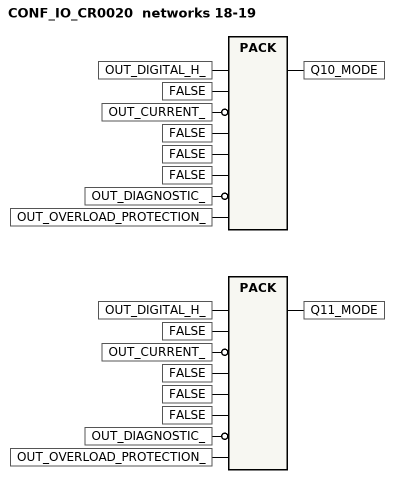
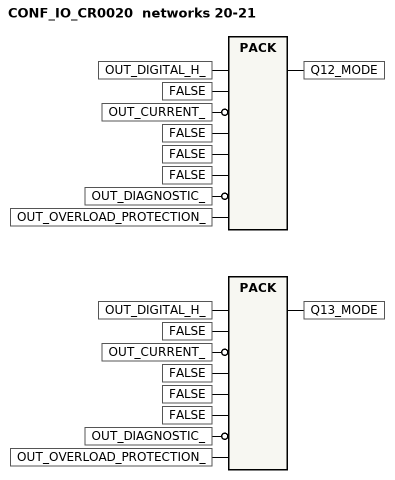
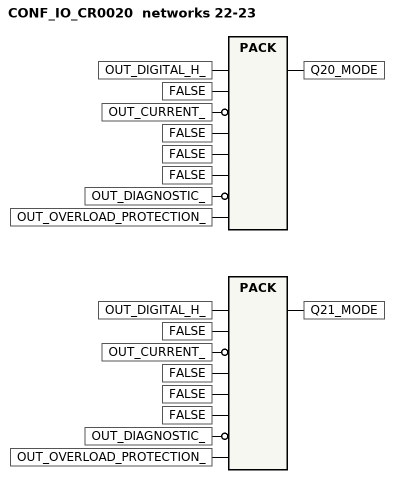
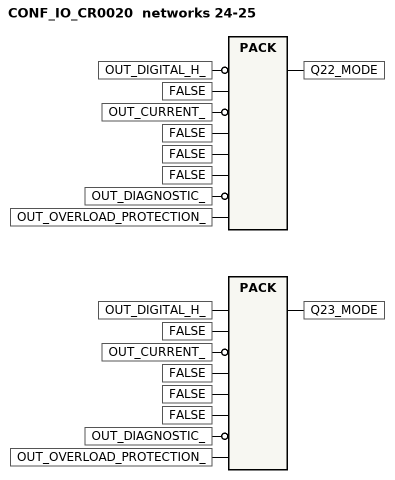
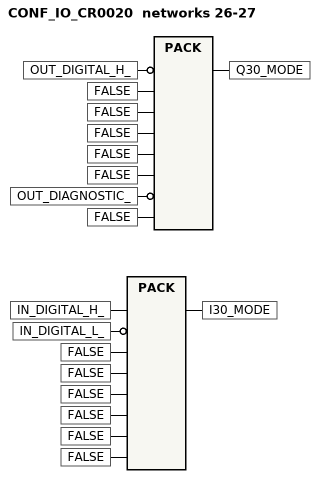
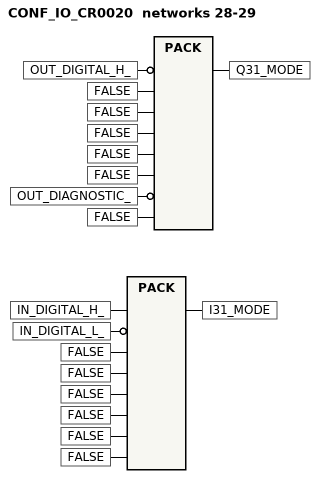
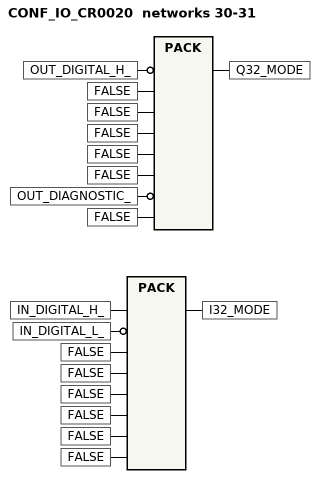
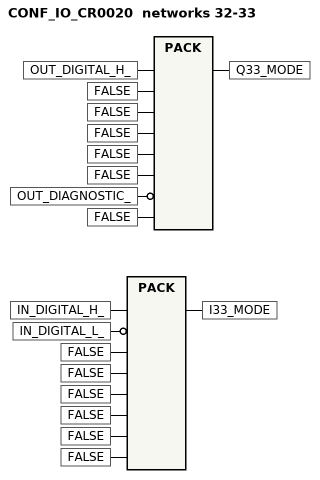
